(* PLC project Unnamed, Unknown Unnamed 1 *)
(* stored: creationDateTime 2020-03-27T18:35:28, modificationDateTime 2020-03-30T18:52:09 *)

(* Function Block Diagram sample *)
PROGRAM program0
  VAR
    LocalVar0 AT %MD0 : DINT := 10;  (* Input 1 *)
    LocalVar1 AT %MD1 : DINT := 20;  (* Input 2 *)
    LocalVar2 AT %MD2 : DINT;  (* Output 1 *)
  END_VAR

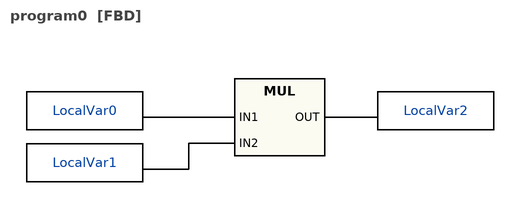
(* FBD diagram, written out as Structured Text *)
LocalVar2 := LocalVar0 * LocalVar1;
END_PROGRAM

CONFIGURATION Config0
  RESOURCE Res0 ON PLC
    TASK task0(INTERVAL := T#1s, PRIORITY := 0);
    PROGRAM instance0 WITH task0 : program0;
  END_RESOURCE
END_CONFIGURATION
